Omron CX-Programmer project NewProject (CX-Programmer 9.03)

# PLC CLP: CJ1M CPU11
I/O table (CPU CJ1M-CPU11): rack 0 slot 0 CJ1W-ETN21(ETN11Mode); rack 0 slot 1 CJ1W-ID211; rack 0 slot 2 CJ1W-OD211; rack 0 slot 3 CJ1W-ID211; rack 0 slot 4 CJ1W-OD211; rack 0 slot 5 CJ1W-ID211; rack 0 slot 6 CJ1W-OD232

## Program NewProgram1 (cyclic task 0)
Local symbols
AS_RS_Ativado 5.02 BOOL
AS_RS_Eixo_X_Ctrg 5.04 BOOL
AS_RS_Eixo_X_D0 5.05 BOOL
AS_RS_Eixo_X_D1 5.06 BOOL
AS_RS_Eixo_X_D2 5.07 BOOL
AS_RS_Eixo_X_D3 5.08 BOOL
AS_RS_Eixo_X_To_Home 5.03 BOOL
AS_RS_Eixo_Y_Ctrg 5.10 BOOL
AS_RS_Eixo_Y_D0 5.11 BOOL
AS_RS_Eixo_Y_D1 5.12 BOOL
AS_RS_Eixo_Y_D2 5.13 BOOL
AS_RS_Eixo_Y_D3 5.14 BOOL
AS_RS_Eixo_Y_To_Home 5.09 BOOL
AS_RS_Eixo_Z_Ctrg 6.00 BOOL
AS_RS_Eixo_Z_D0 6.01 BOOL
AS_RS_Eixo_Z_D1 6.02 BOOL
AS_RS_Eixo_Z_D2 6.03 BOOL
AS_RS_Eixo_Z_D3 6.04 BOOL
AS_RS_Eixo_Z_To_Home 5.15 BOOL
AS_RS_Home_X_Completo 4.05 BOOL
AS_RS_Home_Y_Completo 4.07 BOOL
AS_RS_Home_Z_Completo 4.09 BOOL
AS_RS_Pos_X_Completa 4.04 BOOL
AS_RS_Pos_Y_Completa 4.06 BOOL
AS_RS_Pos_Z_Completa 4.08 BOOL
Confirmacao W4.00 BOOL
Eletroval1 1.06 BOOL
Eletroval2 1.07 BOOL
Eletroval3 1.08 BOOL
Eletroval4 1.09 BOOL
Esteira1 1.00 BOOL
Esteira2 1.01 BOOL
Esteira3 1.02 BOOL
Esteira4 1.03 BOOL
Etapa0 W0.00 BOOL
Etapa1 W0.01 BOOL
Etapa2 W0.02 BOOL
Etapa3 W0.03 BOOL
Etapa4 W0.04 BOOL
Etapa5 W0.05 BOOL
Etapa6 W0.06 BOOL
Etapa7 W0.07 BOOL
Sensor1 0.00 BOOL
Sensor2 0.01 BOOL
Sensor3 0.02 BOOL
Sensor4 0.03 BOOL

### Section Main

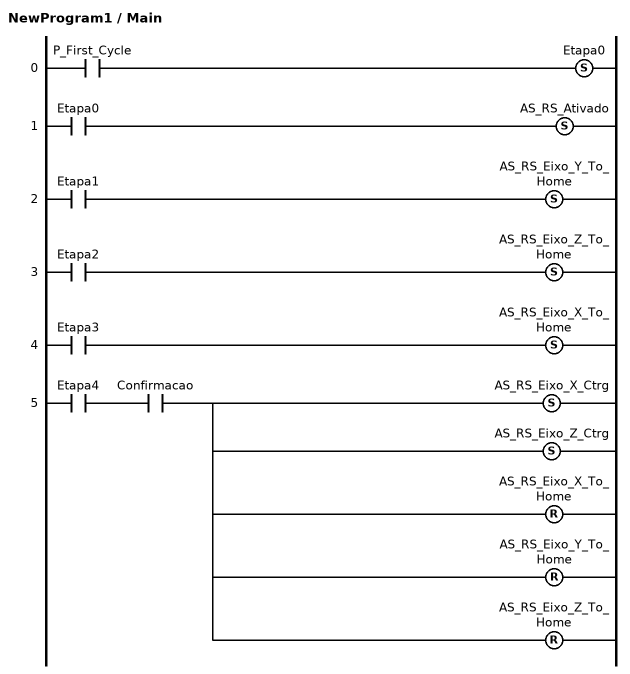
; rung 0
LD P_First_Cycle
SET Etapa0
; rung 1
LD Etapa0
SET AS_RS_Ativado
; rung 2
LD Etapa1
SET AS_RS_Eixo_Y_To_Home
; rung 3
LD Etapa2
SET AS_RS_Eixo_Z_To_Home
; rung 4
LD Etapa3
SET AS_RS_Eixo_X_To_Home
; rung 5
LD Etapa4
AND Confirmacao
SET AS_RS_Eixo_X_Ctrg
SET AS_RS_Eixo_Z_Ctrg
RSET AS_RS_Eixo_X_To_Home
RSET AS_RS_Eixo_Y_To_Home
RSET AS_RS_Eixo_Z_To_Home

### Section Transitions

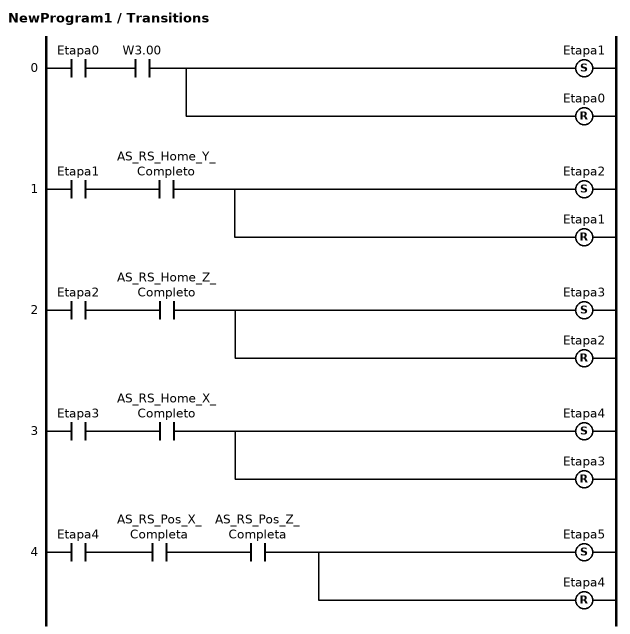
; rung 0
LD Etapa0
AND W3.00
SET Etapa1
RSET Etapa0
; rung 1
LD Etapa1
AND AS_RS_Home_Y_Completo
SET Etapa2
RSET Etapa1
; rung 2
LD Etapa2
AND AS_RS_Home_Z_Completo
SET Etapa3
RSET Etapa2
; rung 3
LD Etapa3
AND AS_RS_Home_X_Completo
SET Etapa4
RSET Etapa3
; rung 4
LD Etapa4
AND AS_RS_Pos_X_Completa
AND AS_RS_Pos_Z_Completa
SET Etapa5
RSET Etapa4

### Section END
; rung 0
END(001)